FUNCTION_BLOCK AllRTUStat
VAR_INPUT
END_VAR
VAR_OUTPUT
END_VAR
VAR_TEMP	
	
	i:INT;
	
END_VAR

//Deci.GVL.nInputCoilIndex      := Lib.GVL_DataHalls.StartInputCoilIndex_RTUStat;
//Deci.GVL.nOutputCoilIndex     := Deci.GVL_DataHalls.StartOutputCoilIndex_RTUStat;
//Deci.GVL.nInputRegisterIndex  := Deci.GVL_DataHalls.StartInputRegisterIndex_RTUStat;
//Deci.GVL.nOutputRegisterIndex := Deci.GVL_DataHalls.StartOutputRegisterIndex_RTUStat;

i:= Lib.GVL.nInputCoilIndex;

Lib.GVL.mb_Input_Coils[i+0] :=  Lib.GVL_THT.THT[1].CommsError;
Lib.GVL.mb_Input_Coils[i+1] :=  Lib.GVL_THT.THT[2].CommsError;
Lib.GVL.mb_Input_Coils[i+2] :=  Lib.GVL_THT.THT[3].CommsError;
Lib.GVL.mb_Input_Coils[i+3] :=  Lib.GVL_THT.THT[4].CommsError;
Lib.GVL.mb_Input_Coils[i+4] :=  Lib.GVL_THT.THT[5].CommsError;
Lib.GVL.mb_Input_Coils[i+5] :=  Lib.GVL_THT.THT[6].CommsError;
Lib.GVL.mb_Input_Coils[i+6] :=  Lib.GVL_THT.THT[7].CommsError;
Lib.GVL.mb_Input_Coils[i+7] :=  Lib.GVL_THT.THT[8].CommsError;
Lib.GVL.mb_Input_Coils[i+8] :=  Lib.GVL_THT.THT[9].CommsError;
Lib.GVL.mb_Input_Coils[i+9] :=  Lib.GVL_THT.THT[10].CommsError;
Lib.GVL.mb_Input_Coils[i+10] := Lib.GVL_THT.THT[11].CommsError;
Lib.GVL.mb_Input_Coils[i+11] := Lib.GVL_THT.THT[12].CommsError;
Lib.GVL.mb_Input_Coils[i+12] := Lib.GVL_THT.THT[13].CommsError;
Lib.GVL.mb_Input_Coils[i+13] := Lib.GVL_THT.THT[14].CommsError;

//Lib.GVL.mb_Input_Coils[i+14] := Lib.GVL_THT.THT[15].CommsError;
//Lib.GVL.mb_Input_Coils[i+15] := Lib.GVL_THT.THT[16].CommsError;

i:=Lib.GVL.nInputRegisterIndex;

Lib.GVL.mb_Input_Registers[i+0]:= INT_TO_WORD(Lib.GVL_THt.THT[1].CommsErrorCode);
Lib.GVL.mb_Input_Registers[i+1]:= INT_TO_WORD(Lib.GVL_THt.THT[2].CommsErrorCode);
Lib.GVL.mb_Input_Registers[i+2]:= INT_TO_WORD(Lib.GVL_THt.THT[3].CommsErrorCode);
Lib.GVL.mb_Input_Registers[i+3]:= INT_TO_WORD(Lib.GVL_THt.THT[4].CommsErrorCode);
Lib.GVL.mb_Input_Registers[i+4]:= INT_TO_WORD(Lib.GVL_THt.THT[5].CommsErrorCode);
Lib.GVL.mb_Input_Registers[i+5]:= INT_TO_WORD(Lib.GVL_THt.THT[6].CommsErrorCode);
Lib.GVL.mb_Input_Registers[i+6]:= INT_TO_WORD(Lib.GVL_THt.THT[7].CommsErrorCode);
Lib.GVL.mb_Input_Registers[i+7]:= INT_TO_WORD(Lib.GVL_THt.THT[8].CommsErrorCode);
Lib.GVL.mb_Input_Registers[i+8]:= INT_TO_WORD(Lib.GVL_THt.THT[9].CommsErrorCode);
Lib.GVL.mb_Input_Registers[i+9]:= INT_TO_WORD(Lib.GVL_THt.THT[10].CommsErrorCode);
Lib.GVL.mb_Input_Registers[i+10]:= INT_TO_WORD(Lib.GVL_THt.THT[11].CommsErrorCode);
Lib.GVL.mb_Input_Registers[i+11]:= INT_TO_WORD(Lib.GVL_THt.THT[12].CommsErrorCode);

Lib.GVL.mb_Input_Registers[i+12]:= INT_TO_WORD(Lib.GVL_THt.THT[13].CommsErrorCode);
Lib.GVL.mb_Input_Registers[i+13]:= INT_TO_WORD(Lib.GVL_THt.THT[14].CommsErrorCode);
//Lib.GVL.mb_Input_Registers[i+14]:= INT_TO_WORD(Lib.GVL_THt.THT[15].CommsErrorCode);

END_FUNCTION_BLOCK

(* stored: Version 1.1.0.1, ProductVersion 3.1.4024.12
   POU AllRTUStat: Id {f82f79bd-b4a5-4084-be1e-8d065e72dbfc}, SpecialFunc None *)
